FUNCTION_BLOCK INTERNAL FB_ChargedState IMPLEMENTS I_State
VAR
	pMachine				: POINTER TO FB_Machine; // Points to the state machine (THIS)	
	fVSensors 				: ARRAY[0..1] OF REAL;
END_VAR

METHOD PUBLIC Check 
VAR
	fInputVoltage			: REAL;
	fLoadVoltage 			: REAL; 
END_VAR
THIS^.SetMainContactors(); // not necessary but reinforces safety 
THIS^.SetBypassContactors(); // necessary

fVSensors := THIS^.pMachine^.VSensors;

fLoadVoltage := fVSensors[1];
fInputVoltage := fVSensors[0];

IF (fLoadVoltage <= 1.1 * fInputVoltage AND fLoadVoltage >= 0.9502 * fInputVoltage) THEN
	IF (fInputVoltage >= THIS^.pMachine^.LowerBoundV AND fInputVoltage <= THIS^.pMachine^.UpperBoundV) THEN
		THIS^.pMachine^.Message := '[CHARGED] The input and load voltages are within the boundaries. $0A PRESS "DISCHARGE" TO ENTER DISCHARGE STATE';
  	ELSE 
		THIS^.pMachine^.Message := '[CHARGED] The load voltage corresponds to the input voltage, but is not included within the defined limits.$0A THE SYSTEM ENTERS DISCHARGE STATE';
		THIS^.pMachine^.SetState(THIS^.pMachine^.DischargeState);
	END_IF
 
ELSE
	THIS^.pMachine^.Message := '[CHARGED] The load voltage DOES NOT match the input voltage.$0A THE SYSTEM ENTERS DISCHARGE STATE';
	THIS^.pMachine^.SetState(THIS^.pMachine^.DischargeState);
END_IF
END_METHOD

PROPERTY PUBLIC Description : STRING
GET
Description := 'CHARGED';
END_GET
END_PROPERTY

METHOD PUBLIC FB_init 
VAR_INPUT
	bInitRetains 	: BOOL; // if TRUE, the retain variables are initialized (warm start / cold start)
	bInCopyCode 	: BOOL;  // if TRUE, the instance afterwards gets moved into the copy code (online change)
	
	pMachine		: POINTER TO FB_Machine; // Points to the state machine (THIS)
END_VAR
THIS^.pMachine := pMachine;
END_METHOD

METHOD PUBLIC PressButton
END_METHOD

METHOD PUBLIC PressDischarge
THIS^.pMachine^.Message := '[CHARGED] Discharge button has been pressed. $0A SYSTEM ENTERS DISCHARGE STATE.';
THIS^.pMachine^.SetState(THIS^.pMachine^.DischargeState);
END_METHOD

METHOD PUBLIC Reset
THIS^.pMachine^.Message := '[CHARGED] Reset button has been pressed. $0A SYSTEM ENTERS DISCHARGE STATE.';
THIS^.pMachine^.SetState(THIS^.pMachine^.DischargeState);
END_METHOD

METHOD PUBLIC SetBypassContactors
VAR
	nIdx				: INT;
	bBypassContactors	: ARRAY[0..1] OF BOOL;
END_VAR
FOR nIdx := 0 TO 1 DO 
	bBypassContactors[nIdx] := TRUE; 
END_FOR

THIS^.pMachine^.BypassContactors := bBypassContactors;
END_METHOD

METHOD PUBLIC SetMainContactors
VAR
	nIdx				: INT;
	bMainContactors 	: ARRAY[0..1] OF BOOL;
END_VAR
FOR nIdx := 0 TO 1 DO 
	bMainContactors[nIdx] := TRUE;
END_FOR

THIS^.pMachine^.MainContactors := bMainContactors;
END_METHOD

METHOD PUBLIC Stop
THIS^.pMachine^.SetState(THIS^.pMachine^.ErrorState);
END_METHOD

METHOD PUBLIC TimerDone
END_METHOD

END_FUNCTION_BLOCK

(* stored: Version 1.1.0.1, ProductVersion 3.1.4024.12
   POU FB_ChargedState: Id {6ccb0767-b26e-4ca8-b32e-b0274bc0898c}, SpecialFunc None
   Method Check: Id {fedb8386-7dee-4770-bcfd-13bf41bd1b84}
   Property Description: Id {fc9f2ec7-d167-4132-9d9f-13de5948a19e}
   Get Get: Id {4e7123ed-cd33-47ab-8743-ade73c3f1c6c}
   Method FB_init: Id {efde9a62-674a-488a-99b1-3c8f9066992d}
   Method PressButton: Id {231f6bc4-0fe7-4fcb-a90e-7626ad2adeb0}
   Method PressDischarge: Id {edac99bf-f040-4eaf-a27a-fdea7a5b1dcc}
   Method Reset: Id {b7743eac-850b-46c9-994c-dc501161fe3b}
   Method SetBypassContactors: Id {e961f1d6-7819-403e-8041-72813777c5e0}
   Method SetMainContactors: Id {3a7a8f7c-ae40-49d5-8840-68e5675f2352}
   Method Stop: Id {00130648-37c2-420d-abb2-efa751e9696b}
   Method TimerDone: Id {2d662e3e-8fd2-498a-9f96-83f3a4fa2ba0} *)
